// TIA Portal V16 export
// export: Created 2024-12-03T15:41:45.3331491Z, ExportSetting WithReadOnly, DisplayName Totally Integrated Automation Portal, DisplayVersion V16 Update 6, DisplayName TIA Portal Version Control Interface, DisplayVersion V16 Update 2, DisplayName TIA Portal Openness, DisplayVersion V16 Update 6, DisplayName TIA Portal Teamcenter Gateway, DisplayVersion V16, DisplayName SINAMICS Startdrive Advanced, DisplayVersion V16 Update 5, DisplayName SINAMICS Startdrive G130, G150, S120, S150, SINAMICS MV, S210, DisplayVersion V16 Update 5, DisplayName SINAMICS Startdrive G110M, G120, G120C, G120D, G120P, G115D, DisplayVersion V16 Update 5, DisplayName STEP 7 Professional, DisplayVersion V16 Update 6, DisplayName STEP 7 Safety, DisplayVersion V16, DisplayName WinCC Advanced / Unified PC, DisplayVersion V16 Update 6
TYPE "COGNEX_DATAMAN_IN_STATUS_UDT"
// stored: CreationDate 2022-02-10T08:20:21.8932261Z, InterfaceModifiedDate 2022-02-10T08:21:09.6700619Z, IsConsistent true, LibraryConformanceStatus The object is library-conformant., ModifiedDate 2022-02-10T08:21:09.6700619Z
   STRUCT
      TriggerReady : Bool;
      TriggerAck : Bool;
      spare2 : Bool;
      MissedAck : Bool;
      spare4 : Bool;
      spare5 : Bool;
      spare6 : Bool;
      spare7 : Bool;
      TriggerId_LSB : Byte;
      TriggerId_MSB : Byte;
   END_STRUCT;
END_TYPE
